// TIA Portal V19 export
TYPE "LAF_typeGlobalDateTime"
TITLE = Structure date&time / Struktur Date&Time
// Type for global date and time, with different formats and return value storage. / Globale Informationen
// stored: Access Published
   STRUCT
      retVal : Int;   // Status Uhrzeit lesen / State read time
      dtl : DTL;   // Datum & Zeit im DTL Format / Date&Time type DTL
      ldt : LDT;   // Date&Time type LDT / Datum & Zeit im LDT Format
      "dt" : Date_And_Time;   // Datum & Zeit im DT Format / Date&Time type DT
   END_STRUCT;
END_TYPE
